{attribute 'qualified_only'}
{attribute 'strict'}
TYPE E_ModuleLevel :
(
	INFO 		:= 0,
	WARNING 	:= 1,
	ALARM		:= 2,
	CRITICAL	:= 3
);
END_TYPE

(* stored: Version 1.1.0.1, ProductVersion 3.1.4024.13
   EnumerationTextList E_ModuleLevel: Id {09ed1a9d-c7e3-46c7-b801-145016d9b09d} *)
